// TIA Portal V21 export
VAR_GLOBAL   // PLC tag table "InputAnalogici_010102"
   LivelloVascaProdotto AT %IW200 : Word;
   Pressione_PR1_IngressoFiltriProdotto AT %IW202 : Word;
   Pressione_PR2_UscitaFiltriProdotto AT %IW204 : Word;
   Portata_FL1_IngressoSterilizzatore AT %IW206 : Word;
   Pressione_PR4_ControPressione_CP1 AT %IW210 : Word;
   Pressione_PR5_ControPressione_CP2 AT %IW212 : Word;
   Temperatura_TC1_UscitaSterilizzatore_Processo AT %IW216 : Word;
   Temperatura_TC2_Scorta AT %IW218 : Word;
   Temperatura_TC3_AcquaCalda AT %IW220 : Word;
   Temperatura_TC4_IngressoSosta AT %IW222 : Word;
   Temperatura_TC5_FineLinea AT %IW224 : Word;
   Temperatura_TC6_UscitaSosta_Processo AT %IW226 : Word;
   Pressione_PR3_SicurezzaIngressoSterilizzatore AT %IW208 : Word;
   Ew214 AT %IW214 : Word;
   Temperatura_TC7_UscitaSterilizzatore_Storicizzazione AT %IW228 : Word;
   Temperatura_TC8_UscitaRaffredatore_Processo AT %IW230 : Word;
   Temperatura_TC9_UscitaSosta_Storicizzazione AT %IW232 : Word;
   Temperatura_TC10_BarriereVapore_ScambioValvole AT %IW234 : Word;
   Temperatura_TC11_BarriereVapore_TuboInTubo AT %IW236 : Word;
   Ew238 AT %IW238 : Word;
END_VAR
